INTERFACE I_StringBuilder

METHOD Append : I_StringBuilder
VAR_INPUT
	sText	: T_MaxString;
END_VAR
END_METHOD

METHOD Reset : I_LimitedStringBuilder
VAR_INPUT
END_VAR
END_METHOD

METHOD ToLowerCase : I_StringBuilder
VAR_INPUT
END_VAR
END_METHOD

METHOD ToString : T_MaxString
VAR_INPUT
END_VAR
END_METHOD

METHOD ToUpperCase : I_StringBuilder
VAR_INPUT
END_VAR
END_METHOD

END_INTERFACE

(* stored: Version 1.1.0.1
   Itf I_StringBuilder: Id {6b364cdd-797f-4330-bd1d-3e4d4a7b2a6d}
   Method Append: Id {f020974a-8325-40d4-8559-0fe02bf4ddfe}
   Method Reset: Id {4545a6ae-d943-4de7-b047-70e643eb9bd6}
   Method ToLowerCase: Id {b0e86b3a-1003-40c0-addd-2d2183df650c}
   Method ToString: Id {5f2a8976-38b0-43b2-9726-0e94f7bc5c25}
   Method ToUpperCase: Id {85955b9d-b68b-47ec-ae6d-aaecbc6d7e1c} *)
